(* CODESYS project Applikation FN Set TSR starpoint.project

Project tree, tasks and I/O mapping:
  XV100 : XV100, Eaton Automation, version 3.5.3.0
    application Application
      libraries: Standard, 3.5.2.0 (System); CAA SerialCom, 3.5.3.0 (CAA Technical Workgroup)
      task Task (cyclic, interval t#10ms, priority 1) calls MAIN
      Symbols
      program MAIN [ST]
      global variables GLOBAL
*)

// XV100/Application/GLOBAL
VAR_GLOBAL
//FB Globale Var
iStartPosx				:INT;		//Die Globale Variable des Neuen nulpunkts für die anderen FB's
iStartPosy				:INT;		//""
END_VAR

// XV100/Application/MAIN
PROGRAM MAIN
VAR
//FB EINGANGS VAR
iStartpointx			:INT;		//Der Virtuelle x Nullpunkt.
iStartpointy			:INT;		//Der Virtuelle y Nullpunkt.
END_VAR

iStartPosx := iStartpointx;			//Speicher eingang in Global Var
iStartPosy := iStartpointy;			//Speicher eingang in Global Var

END_PROGRAM
